// ---- OOPs/FB_HighLevelSystem.TcPOU
FUNCTION_BLOCK FB_HighLevelSystem IMPLEMENTS ITF_HighLevelSystem
VAR_INPUT
	eActivationStatus : ActivationStatus;
END_VAR
VAR_OUTPUT
END_VAR
VAR
END_VAR

PROPERTY eCondition : HighLevelCondition
GET
END_GET
END_PROPERTY

PROPERTY nErrorID : UDINT
GET
END_GET
END_PROPERTY

END_FUNCTION_BLOCK

// ---- POUs/ServiceModule/FB_DistanceSensor.TcPOU
FUNCTION_BLOCK FB_DistanceSensor IMPLEMENTS ITF_SubSystem
VAR_OUTPUT
	fDistance 			: LREAL;
END_VAR
VAR
	//Local
	fbEL6021			: FB_SerialComRS422;

	//ErrorBits
	bCommunicationError : BIT;
	bOutOfRange 		: BIT;
END_VAR
VAR CONSTANT
	fSMR 		: LREAL := 50.0;				// Start of Measuring Range
	fEMR 		: LREAL := 150.0;				// End of Measuring Range
END_VAR

fbEL6021(stReceiveData:=DistanceSensor.stEL6021In, stTransmitData:=DistanceSensor.stEL6021Out);

fDistance := fbEL6021.fDistance;

METHOD PRIVATE doCheckRange : BOOL
VAR_INPUT
	fDistanceValue : LREAL;
	fMax : LREAL;
	fMin : LREAL;
END_VAR
IF fDistanceValue < fMin OR fDistanceValue > fMax THEN
	doCheckRange := FALSE;
	fDistance := 999;
ELSE
	doCheckRange := TRUE;
END_IF
END_METHOD

PROPERTY eCondition : SubLevelCondition
GET
IF nErrorID <> 0 THEN
	eCondition := SubLevelCondition.ERROR;
ELSE
	eCondition := SubLevelCondition.RUN;
END_IF
END_GET
END_PROPERTY

PROPERTY nErrorID : UDINT
GET
IF fbEL6021.eReceiveErrorID <> COMERROR_NOERROR THEN
	bCommunicationError := TRUE;
ELSE
	bCommunicationError := FALSE;
END_IF

bOutOfRange := NOT doCheckRange(fDistanceValue:= fDistance, fMax:=fEMR, fMin:=fSMR);

nErrorID.0 := bCommunicationError;
nErrorID.1 := bOutOfRange;
END_GET
END_PROPERTY

END_FUNCTION_BLOCK

// ---- POUs/ServiceModule/DistanceSensor/FB_SerialComRS422.TcPOU
FUNCTION_BLOCK FB_SerialComRS422
VAR_IN_OUT
	stReceiveData 	: EL6inData22B;
	stTransmitData 	: EL6outData22B;
END_VAR
VAR_OUTPUT
	fDistance : LREAL;
	eReceiveErrorID	: ComError_t;
END_VAR
VAR
	//Receive Buffer
	fbEL6021Ctrl					: SerialLineControl;
	RxBuffer 						: ComBuffer;
	TxBuffer						: ComBuffer;
	//Receive Data
	fbReceiveByte					: ReceiveByte;				
	nFirstThreeBytesOfBuffer  		: ARRAY[0..2] OF BYTE;		// buffer storage for the three bytes that contain the distance information
	nRcvIndex						: UINT := 0;				// Counter
	nDistanceAsStringOfBits			: DINT;
END_VAR
VAR CONSTANT
	fSMR 		: LREAL := 50.0;				// Start of Measuring Range
	fEMR 		: LREAL := 150.0;				// End of Measuring Range
END_VAR

fbEL6021Ctrl(
			Mode:= SERIALLINEMODE_EL6_22B,
			pComIn:= ADR(stReceiveData),
			pComOut:= ADR(stTransmitData),
			SizeComIn:= SIZEOF(stReceiveData),
			Error=>,
			ErrorID=>,
			TxBuffer:=TxBuffer,
			RxBuffer:=RxBuffer,);

fbReceiveByte(RXbuffer := RxBuffer, Error => eReceiveErrorID);

WHILE fbReceiveByte.ByteReceived AND (nRcvIndex <= SIZEOF(nFirstThreeBytesOfBuffer)) DO
	fbReceiveByte(RXbuffer := RxBuffer);
	IF (fbReceiveByte.ReceivedByte.7) = 0 THEN
		nFirstThreeBytesOfBuffer[nRcvIndex] := fbReceiveByte.ReceivedByte;
		nRcvIndex := nRcvIndex + 1;
	ELSE
		nFirstThreeBytesOfBuffer[2] := fbReceiveByte.ReceivedByte;
		nRcvIndex	:= 0;
	END_IF
END_WHILE

doSortBits(nByteBuffer:=nFirstThreeBytesOfBuffer);
doConvertToDistanceValue(nBitString:=nDistanceAsStringOfBits, fMax:=fEMR, fMin:=fSMR);

METHOD PRIVATE doConvertToDistanceValue
VAR_INPUT
	nBitString : DINT;
	fMax : LREAL;
	fMIn : LREAL;
END_VAR
fDistance := 50.0 + 1.0/100.0 * (102.0/65520.0 * DINT_TO_LREAL(nBitString) - 1.0) * (fMax - fMIn);
END_METHOD

METHOD PRIVATE doSortBits
VAR_INPUT
	nByteBuffer : ARRAY [0..2] OF BYTE;
END_VAR
// Rearrange L,M,H Refer Pg 85. We seperate the distance bits from the error, transmissions, ect. -bits in this step.
// MemCopy is a possilbe way to simplify code. But since we need to work with bit and not buyts, this is actually the more readable code.
// Also TwinCAT demands CONST values when working with bit handeling, so loops are also not possible.
nDistanceAsStringOfBits.0 	:= nByteBuffer[0].0;
nDistanceAsStringOfBits.1 	:= nByteBuffer[0].1;
nDistanceAsStringOfBits.2 	:= nByteBuffer[0].2;
nDistanceAsStringOfBits.3 	:= nByteBuffer[0].3;
nDistanceAsStringOfBits.4 	:= nByteBuffer[0].4;
nDistanceAsStringOfBits.5 	:= nByteBuffer[0].5;
nDistanceAsStringOfBits.6 	:= nByteBuffer[1].0;
nDistanceAsStringOfBits.7 	:= nByteBuffer[1].1;
nDistanceAsStringOfBits.8 	:= nByteBuffer[1].2;
nDistanceAsStringOfBits.9 	:= nByteBuffer[1].3;
nDistanceAsStringOfBits.10 	:= nByteBuffer[1].4;
nDistanceAsStringOfBits.11	:= nByteBuffer[1].5;
nDistanceAsStringOfBits.12 	:= nByteBuffer[2].0;
nDistanceAsStringOfBits.13 	:= nByteBuffer[2].1;
nDistanceAsStringOfBits.14 	:= nByteBuffer[2].2;
nDistanceAsStringOfBits.15 	:= nByteBuffer[2].3;
END_METHOD

END_FUNCTION_BLOCK

// ---- POUs/ServiceModule/FB_BoxLED.TcPOU
FUNCTION_BLOCK FB_BoxLED IMPLEMENTS ITF_SubSystem
VAR_INPUT
	eMode : LEDMode;
END_VAR
VAR
	//Local
	nBoxLED : INT;
	fbFlashingTimer : TON;
	bOn : BOOL;
	
	aErrorTimer : ARRAY [0..1] OF TON;
	
	//ErrorBits
	bTemperatureTooHigh : BIT;
	bNoSupplyVoltage : BIT;
END_VAR
VAR CONSTANT
	nIntensity : INT := 32767;				//Intensity [0..32767]
	fDimFactor : REAL := 0.01;				//Percentage (0..100%)
	tSlowFlashingTime : TIME := T#1S;		
	tFastFlashingTime : TIME := T#100MS;
END_VAR

CASE eMode OF
	LEDMode.Off:
			doTurnOn(nBrightness := 0);
	LEDMode.On:
			doTurnOn(nBrightness := nIntensity);
	LEDMode.Dimmed:
			doDimming(fDimmingFactor:=fDimFactor);
	LEDMode.SlowFlashing:
			doFlashing(tFlashingTime:=tSlowFlashingTime);
	LEDMode.FastFlashing:
			doFlashing(tFlashingTime:=tFastFlashingTime);
END_CASE

doSetClampValues();
doGetClampValues();

METHOD PRIVATE doDimming
VAR_INPUT
	fDimmingFactor : REAL;
END_VAR
nBoxLED := REAL_TO_INT(fDimmingFactor * nIntensity);
END_METHOD

METHOD PRIVATE doFlashing
VAR_INPUT
	tFlashingTime : TIME;
END_VAR
fbFlashingTimer(IN:=TRUE, PT:=tFlashingTime);
IF fbFlashingTimer.Q THEN
	fbFlashingTimer(IN:=FALSE);
	bOn := NOT bOn;	
END_IF
IF bOn THEN
	nBoxLED := nIntensity;
ELSE
	nBoxLED := 0;
END_IF
END_METHOD

METHOD PRIVATE doGetClampValues
bTemperatureTooHigh := BoxLED.bBoxGreenWarning;
bNoSupplyVoltage := BoxLED.bBoxGreenError;
END_METHOD

METHOD PRIVATE doSetClampValues
BoxLED.nBoxGreen := nBoxLED;
END_METHOD

METHOD PRIVATE doTurnOn
VAR_INPUT
	nBrightness : INT;
END_VAR
nBoxLED := nBrightness;
END_METHOD

PROPERTY eCondition : SubLevelCondition
GET
IF nErrorID <> 0 THEN
	eCondition := SubLevelCondition.ERROR;
ELSE
	eCondition := SubLevelCondition.RUN;
END_IF
END_GET
END_PROPERTY

PROPERTY nErrorID : UDINT
GET
nErrorID.0 := aErrorTimer[0].Q;
nErrorID.1 := aErrorTimer[1].Q;

aErrorTimer[0](IN := bTemperatureTooHigh, PT := T#5S);
aErrorTimer[1](IN := bNoSupplyVoltage, PT := T#5S);
END_GET
END_PROPERTY

END_FUNCTION_BLOCK

// ---- POUs/ServiceModule/FB_RGBLED.TcPOU
FUNCTION_BLOCK FB_RGBLED IMPLEMENTS ITF_SubSystem
VAR_INPUT
	eColor : LEDColor;
END_VAR
VAR
	//Local
	nRedLED : INT;
	nGreenLED : INT;
	nBlueLED : INT;
	
	aErrorTimer : ARRAY [0..5] OF TON;
	
	//ErrorBits
	bRedTemperatureTooHigh : BIT;
	bRedNoSupplyVoltage : BIT;
	bGreenTemperatureTooHigh : BIT;
	bGreenNoSupplyVoltage : BIT;
	bBlueTemperatureTooHigh : BIT;
	bBlueNoSupplyVoltage : BIT;	
END_VAR
VAR CONSTANT
	nMax : INT := 32767;		//Maximum Intensity (100%)
	nMin : INT := 0;			//Off (0%)
END_VAR

CASE eColor OF
	LEDColor.Off:
		nRedLED := nMin;
		nGreenLED := nMin;
		nBlueLED := nMin;
	LEDColor.Red:
		nRedLED := nMax;
		nGreenLED := nMin;
		nBlueLED := nMin;
	LEDColor.Green:
		nRedLED := nMin;
		nGreenLED := nMax;
		nBlueLED := nMin;
	LEDColor.Blue:
		nRedLED := nMin;
		nGreenLED := nMin;
		nBlueLED := nMax;
END_CASE



doSetClampValues();
doGetClampValues();

METHOD PRIVATE doGetClampValues
VAR_INPUT
END_VAR
bRedTemperatureTooHigh := RGBLED.bRedWarning;
bRedNoSupplyVoltage := RGBLED.bRedError;
bGreenTemperatureTooHigh := RGBLED.bGreenWarning;
bGreenNoSupplyVoltage := RGBLED.bGreenError;
bBlueTemperatureTooHigh := RGBLED.bBlueWarning;
bBlueNoSupplyVoltage := RGBLED.bBlueError;
END_METHOD

METHOD PRIVATE doSetClampValues
RGBLED.nRed := nRedLED;
RGBLED.nGreen := nGreenLED;
RGBLED.nBlue := nBlueLED;
END_METHOD

PROPERTY eCondition : SubLevelCondition
GET
IF nErrorID <> 0 THEN
	eCondition := SubLevelCondition.ERROR;
ELSE
	eCondition := SubLevelCondition.RUN;
END_IF
END_GET
END_PROPERTY

PROPERTY nErrorID : UDINT
GET
nErrorID.0 := aErrorTimer[0].Q;
nErrorID.1 := aErrorTimer[1].Q;
nErrorID.2 := aErrorTimer[2].Q;
nErrorID.3 := aErrorTimer[3].Q;
nErrorID.4 := aErrorTimer[4].Q;
nErrorID.5 := aErrorTimer[5].Q;

aErrorTimer[0](IN:=bRedTemperatureTooHigh, PT:=T#5S);
aErrorTimer[1](IN:=bRedNoSupplyVoltage, PT:=T#5S);
aErrorTimer[2](IN:=bGreenTemperatureTooHigh, PT:=T#5S);
aErrorTimer[3](IN:=bGreenNoSupplyVoltage, PT:=T#5S);
aErrorTimer[4](IN:=bBlueTemperatureTooHigh, PT:=T#5S);
aErrorTimer[5](IN:=bBlueNoSupplyVoltage, PT:=T#5S);
END_GET
END_PROPERTY

END_FUNCTION_BLOCK

// ---- POUs/FB_LevitationSystem.TcPOU
FUNCTION_BLOCK FB_LevitationSystem EXTENDS FB_HighLevelSystem
VAR_INPUT
	eState : LevitationSystemSTM;
	nTGControlOption : USINT;
	//eActivationStatus : ActivationStatus;
END_VAR
VAR_OUTPUT
	bEnableCurrentController : BOOL;
	bEnableIControl : BOOL;
	bEnablePControl : BOOL;
END_VAR
VAR
	fbEqualizingControl			: FB_EqualizingController;
	fbTrajectoryGeneratorXMC1	: FB_TrajectoryGenerator;
	fbTrajectoryGeneratorXMC2	: FB_TrajectoryGenerator;
	fbTrajectoryGeneratorXMC3	: FB_TrajectoryGenerator;
	fbTrajectoryGeneratorXMC4	: FB_TrajectoryGenerator;
	
	fActualLevDistanceForFmag : ARRAY [0..3] OF REAL;
	fActualLevCurrentForFmag : ARRAY [0..3] OF REAL;
	
	fDesiredLevDistance : REAL;
END_VAR

IF eActivationStatus = ActivationStatus.Enabled THEN
	//High Level State Machine
	CASE eState OF
		LevitationSystemSTM.Idling:
			;
			
			
		LevitationSystemSTM.Stationary:
			bEnableCurrentController := FALSE;
			fbTrajectoryGeneratorXMC1.bTransition := FALSE;
			fbTrajectoryGeneratorXMC2.bTransition := FALSE;
			fbTrajectoryGeneratorXMC3.bTransition := FALSE;
			fbTrajectoryGeneratorXMC4.bTransition := FALSE;

			fbEqualizingControl.bActive := FALSE;		
		
			doSetOperationMode();
			
			fbTrajectoryGeneratorXMC1();
			fbTrajectoryGeneratorXMC2();
			fbTrajectoryGeneratorXMC3();
			fbTrajectoryGeneratorXMC4();
			fbEqualizingControl();
			
		LevitationSystemSTM.Transitioning:
			bEnableCurrentController := TRUE;
//			fbTrajectoryGeneratorXMC1.bTransition := TRUE;
//			fbTrajectoryGeneratorXMC2.bTransition := TRUE;
//			fbTrajectoryGeneratorXMC3.bTransition := TRUE;
//			fbTrajectoryGeneratorXMC4.bTransition := TRUE;
			
			//optional AirGap Check to go back into Transition		
			IF fActualLevDistanceForFmag[0] <> fDesiredLevDistance THEN
				fbTrajectoryGeneratorXMC1.bTransition := TRUE;
			ELSE
				fbTrajectoryGeneratorXMC1.bTransition := FALSE;
			END_IF
			IF fActualLevDistanceForFmag[1] <> fDesiredLevDistance THEN
				fbTrajectoryGeneratorXMC2.bTransition := TRUE;
			ELSE
				fbTrajectoryGeneratorXMC2.bTransition := FALSE;
			END_IF
			IF fActualLevDistanceForFmag[2] <> fDesiredLevDistance THEN
				fbTrajectoryGeneratorXMC3.bTransition := TRUE;
			ELSE
				fbTrajectoryGeneratorXMC3.bTransition := FALSE;
			END_IF
			IF fActualLevDistanceForFmag[3] <> fDesiredLevDistance THEN
				fbTrajectoryGeneratorXMC4.bTransition := TRUE;
			ELSE
				fbTrajectoryGeneratorXMC4.bTransition := FALSE;
			END_IF
			
			fbEqualizingControl.bActive := FALSE;
			
			fbTrajectoryGeneratorXMC1();
			fbTrajectoryGeneratorXMC2();
			fbTrajectoryGeneratorXMC3();
			fbTrajectoryGeneratorXMC4();
			fbEqualizingControl();
			
			
		LevitationSystemSTM.HoldingAirGap:
			bEnableCurrentController := FALSE;
			fbTrajectoryGeneratorXMC1.bTransition := FALSE;
			fbTrajectoryGeneratorXMC2.bTransition := FALSE;
			fbTrajectoryGeneratorXMC3.bTransition := FALSE;
			fbTrajectoryGeneratorXMC4.bTransition := FALSE;
			
			fbEqualizingControl.bActive := TRUE;
			
			doCalculateFmagValuesForEC(	fActualLevDistance := fActualLevDistanceForFmag,			//to be implemented
										fActualCurrent := fActualLevCurrentForFmag);
			
			fbTrajectoryGeneratorXMC1();
			fbTrajectoryGeneratorXMC2();
			fbTrajectoryGeneratorXMC3();
			fbTrajectoryGeneratorXMC4();
			fbEqualizingControl();
			
			
		LevitationSystemSTM.TransitioningToZero:
			bEnableCurrentController := TRUE;
			fbTrajectoryGeneratorXMC1.bTransition := TRUE;
			fbTrajectoryGeneratorXMC2.bTransition := TRUE;
			fbTrajectoryGeneratorXMC3.bTransition := TRUE;
			fbTrajectoryGeneratorXMC4.bTransition := TRUE;
			
			fbEqualizingControl.bActive := FALSE;
			
			doSetPresetTGValuesForBackToGround();		//to be implemented with Controller structure
			
			fbTrajectoryGeneratorXMC1();
			fbTrajectoryGeneratorXMC2();
			fbTrajectoryGeneratorXMC3();
			fbTrajectoryGeneratorXMC4();
			fbEqualizingControl();
			
	END_CASE	

END_IF

PROPERTY PUBLIC aECOutputZVector : ARRAY [0..3] OF REAL
GET
aECOutputZVector[0] := fbEqualizingControl.fdzVector[0];
aECOutputZVector[1] := fbEqualizingControl.fdzVector[1];
aECOutputZVector[2] := fbEqualizingControl.fdzVector[2];
aECOutputZVector[3] := fbEqualizingControl.fdzVector[3];
END_GET
END_PROPERTY

PROPERTY PUBLIC aTGActualLevAcceleration : ARRAY [0..3] OF REAL
SET
fbTrajectoryGeneratorXMC1.fInitialAcceleration := aTGActualLevAcceleration[0];
fbTrajectoryGeneratorXMC2.fInitialAcceleration := aTGActualLevAcceleration[1];
fbTrajectoryGeneratorXMC3.fInitialAcceleration := aTGActualLevAcceleration[2];
fbTrajectoryGeneratorXMC4.fInitialAcceleration := aTGActualLevAcceleration[3];
END_SET
END_PROPERTY

PROPERTY PUBLIC aTGActualLevCurrent : ARRAY [0..3] OF REAL
SET
fActualLevCurrentForFmag := aTGActualLevCurrent;

fbTrajectoryGeneratorXMC1.fInitialCurrent := aTGActualLevCurrent[0];
fbTrajectoryGeneratorXMC2.fInitialCurrent := aTGActualLevCurrent[1];
fbTrajectoryGeneratorXMC3.fInitialCurrent := aTGActualLevCurrent[2];
fbTrajectoryGeneratorXMC4.fInitialCurrent := aTGActualLevCurrent[3];
END_SET
END_PROPERTY

PROPERTY PUBLIC aTGActualLevDistance : ARRAY [0..3] OF REAL
SET
fActualLevDistanceForFmag := aTGActualLevDistance;

fbTrajectoryGeneratorXMC1.fInitialAirGap := aTGActualLevDistance[0];
fbTrajectoryGeneratorXMC2.fInitialAirGap := aTGActualLevDistance[1];
fbTrajectoryGeneratorXMC3.fInitialAirGap := aTGActualLevDistance[2];
fbTrajectoryGeneratorXMC4.fInitialAirGap := aTGActualLevDistance[3];
END_SET
END_PROPERTY

PROPERTY PUBLIC aTGActualLevVelocity : ARRAY [0..3] OF REAL
SET
fbTrajectoryGeneratorXMC1.fInitialVelocity := aTGActualLevVelocity[0];
fbTrajectoryGeneratorXMC2.fInitialVelocity := aTGActualLevVelocity[1];
fbTrajectoryGeneratorXMC3.fInitialVelocity := aTGActualLevVelocity[2];
fbTrajectoryGeneratorXMC4.fInitialVelocity := aTGActualLevVelocity[3];
END_SET
END_PROPERTY

PROPERTY PUBLIC aTGOutputLevAcceleration : ARRAY [0..3] OF REAL
GET
aTGOutputLevAcceleration[0] := fbTrajectoryGeneratorXMC1.fNewReferenceValueForAcceleration;
aTGOutputLevAcceleration[1] := fbTrajectoryGeneratorXMC2.fNewReferenceValueForAcceleration;
aTGOutputLevAcceleration[2] := fbTrajectoryGeneratorXMC3.fNewReferenceValueForAcceleration;
aTGOutputLevAcceleration[3] := fbTrajectoryGeneratorXMC4.fNewReferenceValueForAcceleration;
END_GET
END_PROPERTY

PROPERTY PUBLIC aTGOutputLevCurrent : ARRAY [0..3] OF REAL
GET
aTGOutputLevCurrent[0] := fbTrajectoryGeneratorXMC1.fNewReferenceValueForCurrent;
aTGOutputLevCurrent[1] := fbTrajectoryGeneratorXMC2.fNewReferenceValueForCurrent;
aTGOutputLevCurrent[2] := fbTrajectoryGeneratorXMC3.fNewReferenceValueForCurrent;
aTGOutputLevCurrent[3] := fbTrajectoryGeneratorXMC4.fNewReferenceValueForCurrent;
END_GET
END_PROPERTY

PROPERTY PUBLIC aTGOutputLevDistance : ARRAY [0..3] OF REAL
GET
aTGOutputLevDistance[0] := fbTrajectoryGeneratorXMC1.fNewReferenceValueForAirGap;
aTGOutputLevDistance[1] := fbTrajectoryGeneratorXMC2.fNewReferenceValueForAirGap;
aTGOutputLevDistance[2] := fbTrajectoryGeneratorXMC3.fNewReferenceValueForAirGap;
aTGOutputLevDistance[3] := fbTrajectoryGeneratorXMC4.fNewReferenceValueForAirGap;
END_GET
END_PROPERTY

PROPERTY PUBLIC aTGOutputLevForce : ARRAY [0..3] OF REAL
GET
aTGOutputLevForce[0] := fbTrajectoryGeneratorXMC1.fNewReferenceValueForForce;
aTGOutputLevForce[1] := fbTrajectoryGeneratorXMC2.fNewReferenceValueForForce;
aTGOutputLevForce[2] := fbTrajectoryGeneratorXMC3.fNewReferenceValueForForce;
aTGOutputLevForce[3] := fbTrajectoryGeneratorXMC4.fNewReferenceValueForForce;
END_GET
END_PROPERTY

PROPERTY PUBLIC aTGOutputLevVelocity : ARRAY [0..3] OF REAL
GET
aTGOutputLevVelocity[0] := fbTrajectoryGeneratorXMC1.fNewReferenceVaueForVelocity;
aTGOutputLevVelocity[1] := fbTrajectoryGeneratorXMC2.fNewReferenceVaueForVelocity;
aTGOutputLevVelocity[2] := fbTrajectoryGeneratorXMC3.fNewReferenceVaueForVelocity;
aTGOutputLevVelocity[3] := fbTrajectoryGeneratorXMC4.fNewReferenceVaueForVelocity;
END_GET
END_PROPERTY

PROPERTY PUBLIC aTGOutputLevVoltage : ARRAY [0..3] OF REAL
GET
aTGOutputLevVoltage[0] := fbTrajectoryGeneratorXMC1.fNewReferenceValueForVoltage;
aTGOutputLevVoltage[1] := fbTrajectoryGeneratorXMC2.fNewReferenceValueForVoltage;
aTGOutputLevVoltage[2] := fbTrajectoryGeneratorXMC3.fNewReferenceValueForVoltage;
aTGOutputLevVoltage[3] := fbTrajectoryGeneratorXMC4.fNewReferenceValueForVoltage;
END_GET
END_PROPERTY

PROPERTY PUBLIC bTrajectoryCompleted : BOOL
GET
VAR
	bTrajectoryCompletedXMC1 : BOOL;
	bTrajectoryCompletedXMC2 : BOOL;
	bTrajectoryCompletedXMC3 : BOOL;
	bTrajectoryCompletedXMC4 : BOOL;
END_VAR
bTrajectoryCompletedXMC1 := fbTrajectoryGeneratorXMC1.bTrajectoryCompleted;
bTrajectoryCompletedXMC2 := fbTrajectoryGeneratorXMC2.bTrajectoryCompleted;
bTrajectoryCompletedXMC3 := fbTrajectoryGeneratorXMC3.bTrajectoryCompleted;
bTrajectoryCompletedXMC4 := fbTrajectoryGeneratorXMC4.bTrajectoryCompleted;

IF bTrajectoryCompletedXMC1 AND bTrajectoryCompletedXMC2 AND bTrajectoryCompletedXMC3 AND bTrajectoryCompletedXMC4 THEN
	bTrajectoryCompleted := TRUE;
ELSE
	bTrajectoryCompleted := FALSE;
END_IF
END_GET
END_PROPERTY

METHOD PRIVATE doCalculateFmagValuesForEC
VAR_INPUT
	fActualLevDistance : ARRAY [0..3] OF REAL;
	fActualCurrent		: ARRAY [0..3] OF REAL;
END_VAR
fbEqualizingControl.fActualDeltaFmag := 0;
END_METHOD

METHOD PRIVATE doSetOperationMode
VAR_INPUT
END_VAR
IF nTGControlOption.0 THEN
	fbTrajectoryGeneratorXMC1.eMode := TGControllerMode.IControl;
	fbTrajectoryGeneratorXMC2.eMode := TGControllerMode.IControl;
	fbTrajectoryGeneratorXMC3.eMode := TGControllerMode.IControl;
	fbTrajectoryGeneratorXMC4.eMode := TGControllerMode.IControl;
	
	bEnableIControl := TRUE;
	bEnablePControl := FALSE;
END_IF

IF nTGControlOption.1 THEN
	fbTrajectoryGeneratorXMC1.eMode := TGControllerMode.PControl;
	fbTrajectoryGeneratorXMC2.eMode := TGControllerMode.PControl;
	fbTrajectoryGeneratorXMC3.eMode := TGControllerMode.PControl;
	fbTrajectoryGeneratorXMC4.eMode := TGControllerMode.PControl;
	
	bEnableIControl := FALSE;
	bEnablePControl := TRUE;
END_IF
END_METHOD

METHOD PRIVATE doSetPresetTGValuesForBackToGround
VAR_INPUT
END_VAR
END_METHOD

PROPERTY eCondition : HighLevelCondition
GET
IF eActivationStatus = ActivationStatus.Disabled THEN
	eCondition := HighLevelCondition.SLEEP;
ELSE
	IF fbTrajectoryGeneratorXMC1.eCondition = SubLevelCondition.RUN AND fbTrajectoryGeneratorXMC2.eCondition = SubLevelCondition.RUN AND fbTrajectoryGeneratorXMC3.eCondition = SubLevelCondition.RUN AND fbTrajectoryGeneratorXMC4.eCondition = SubLevelCondition.RUN AND fbEqualizingControl.eCondition = SubLevelCondition.RUN THEN
		eCondition := HighLevelCondition.RUN;
	ELSE
		eCondition := HighLevelCondition.INIT;
	END_IF
END_IF
END_GET
END_PROPERTY

PROPERTY PUBLIC fTGDesiredLevAcceleration : REAL
SET
fbTrajectoryGeneratorXMC1.fDesiredAccelerationAfterTransitioning := fTGDesiredLevAcceleration;
fbTrajectoryGeneratorXMC2.fDesiredAccelerationAfterTransitioning := fTGDesiredLevAcceleration;
fbTrajectoryGeneratorXMC3.fDesiredAccelerationAfterTransitioning := fTGDesiredLevAcceleration;
fbTrajectoryGeneratorXMC4.fDesiredAccelerationAfterTransitioning := fTGDesiredLevAcceleration;
END_SET
END_PROPERTY

PROPERTY PUBLIC fTGDesiredLevDistance : REAL
SET
fbTrajectoryGeneratorXMC1.fDesiredAirGapAfterTransitioning := fTGDesiredLevDistance;
fbTrajectoryGeneratorXMC2.fDesiredAirGapAfterTransitioning := fTGDesiredLevDistance;
fbTrajectoryGeneratorXMC3.fDesiredAirGapAfterTransitioning := fTGDesiredLevDistance;
fbTrajectoryGeneratorXMC4.fDesiredAirGapAfterTransitioning := fTGDesiredLevDistance;

fDesiredLevDistance := fTGDesiredLevDistance;
END_SET
END_PROPERTY

PROPERTY PUBLIC fTGDesiredLevTime : REAL
SET
fbTrajectoryGeneratorXMC1.tDesiredTimeForTransitioning := REAL_TO_TIME(fTGDesiredLevTime);
fbTrajectoryGeneratorXMC2.tDesiredTimeForTransitioning := REAL_TO_TIME(fTGDesiredLevTime);
fbTrajectoryGeneratorXMC3.tDesiredTimeForTransitioning := REAL_TO_TIME(fTGDesiredLevTime);
fbTrajectoryGeneratorXMC4.tDesiredTimeForTransitioning := REAL_TO_TIME(fTGDesiredLevTime);
END_SET
END_PROPERTY

PROPERTY PUBLIC fTGDesiredLevVelocity : REAL
SET
fbTrajectoryGeneratorXMC1.fDesiredVelocityAfterTransitioning := fTGDesiredLevVelocity;
fbTrajectoryGeneratorXMC2.fDesiredVelocityAfterTransitioning := fTGDesiredLevVelocity;
fbTrajectoryGeneratorXMC3.fDesiredVelocityAfterTransitioning := fTGDesiredLevVelocity;
fbTrajectoryGeneratorXMC4.fDesiredVelocityAfterTransitioning := fTGDesiredLevVelocity;
END_SET
END_PROPERTY

PROPERTY nErrorID : UDINT
GET
VAR
	nErrorBitsTG1 : UDINT;
	nErrorBitsTG2 : UDINT;
	nErrorBitsTG3 : UDINT;
	nErrorBitsTG4 : UDINT;
	nErrorBitsEC	: UDINT;
END_VAR
nErrorBitsTG1 := fbTrajectoryGeneratorXMC1.nErrorID;
nErrorBitsTG2 := fbTrajectoryGeneratorXMC2.nErrorID;
nErrorBitsTG3 := fbTrajectoryGeneratorXMC3.nErrorID;
nErrorBitsTG4 := fbTrajectoryGeneratorXMC4.nErrorID;
nErrorBitsEC := fbEqualizingControl.nErrorID;


nErrorID.0 := nErrorBitsEC.0;
nErrorID.1 := nErrorBitsEC.1;
nErrorID.2 := nErrorBitsTG1.0;
nErrorID.3 := nErrorBitsTG1.1;
nErrorID.4 := nErrorBitsTG1.2;
nErrorID.5 := nErrorBitsTG1.3;
nErrorID.6 := nErrorBitsTG1.4;
nErrorID.7 := nErrorBitsTG1.5;
nErrorID.8 := nErrorBitsTG2.0;
nErrorID.9 := nErrorBitsTG2.1;
nErrorID.10 := nErrorBitsTG2.2;
nErrorID.11 := nErrorBitsTG2.3;
nErrorID.12 := nErrorBitsTG2.4;
nErrorID.13 := nErrorBitsTG2.5;
nErrorID.14 := nErrorBitsTG3.0;
nErrorID.15 := nErrorBitsTG3.1;
nErrorID.16 := nErrorBitsTG3.2;
nErrorID.17 := nErrorBitsTG3.3;
nErrorID.18 := nErrorBitsTG3.4;
nErrorID.19 := nErrorBitsTG3.5;
nErrorID.20 := nErrorBitsTG4.0;
nErrorID.21 := nErrorBitsTG4.1;
nErrorID.22 := nErrorBitsTG4.2;
nErrorID.23 := nErrorBitsTG4.3;
nErrorID.24 := nErrorBitsTG4.4;
nErrorID.25 := nErrorBitsTG4.5;
END_GET
END_PROPERTY

END_FUNCTION_BLOCK

// ---- POUs/Levitation/FB_EqualizingController.TcPOU
FUNCTION_BLOCK FB_EqualizingController IMPLEMENTS ITF_SubSystem
VAR_INPUT
	fActualDeltaFmag : REAL;
	bActive : BOOL;
END_VAR
VAR_OUTPUT 
	fdzVector : ARRAY [0..3] OF REAL;
END_VAR
VAR
	//Local
	fbPIDController : FB_BasicPID;
	fPIDOutput : LREAL;
	nPIDErrorID : UINT;

	//Error Bits
	bInvalidParamters : BIT;
	bInvalidCycleTime : BIT;
END_VAR
VAR CONSTANT
	//PID paramters
	fSetpointValue : REAL := 0; 			// Reference delta F = 0 N
	fCtrlCycleTime : REAL := 0.1; 			// Update cycle time of PID block
	fKp : REAL := 0.001;  					// Proportional gain of PID block
	fTn : REAL := 1/INT_TO_REAL(150); 
	fTv : REAL := 0;
	fTd : REAL := 0;
	//Saturation parameters
	fdzMax : REAL := 0.001;
	fdzMin : REAL := -0.001;
END_VAR

IF bActive THEN
	fbPIDController(fSetpointValue := fSetpointValue,
					fActualValue := fActualDeltaFmag,
					bReset := NOT bActive,
					fCtrlCycleTime := fCtrlCycleTime,
					fKp := fKp,
					fTn := fTn,
					fTv := fTv,
					fTd := fTd,
					fCtrlOutput => fPIDOutput, nErrorStatus => nPIDErrorID);

					
	// Update the dz output vector
	fdzVector[0] := (-1/INT_TO_REAL(7900))* LREAL_TO_REAL(fPIDOutput);
	fdzVector[1] := (1/INT_TO_REAL(7900))* LREAL_TO_REAL(fPIDOutput);
	fdzVector[2] := (-1/INT_TO_REAL(7900))* LREAL_TO_REAL(fPIDOutput);
	fdzVector[3] := (1/INT_TO_REAL(7900))* LREAL_TO_REAL(fPIDOutput);	  
	
	
	// Saturate the dz output vector
	IF fdzVector[0] > fdzMax THEN
		fdzVector[0] := fdzMax;
	ELSIF fdzVector[0] < fdzMin THEN
		fdzVector[0] := fdzMin;
	END_IF
	
	IF fdzVector[1] > fdzMax THEN
		fdzVector[1] := fdzMax;
	ELSIF fdzVector[1] < fdzMin THEN
		fdzVector[1] := fdzMin;
	END_IF
	
	IF fdzVector[2] > fdzMax THEN
		fdzVector[2] := fdzMax;
	ELSIF fdzVector[2] < fdzMin THEN
		fdzVector[2] := fdzMin;
	END_IF
	
	IF fdzVector[3] > fdzMax THEN
		fdzVector[3] := fdzMax;
	ELSIF fdzVector[3] < fdzMin THEN
		fdzVector[3] := fdzMin;
	END_IF
	
ELSE
	fdzVector[0] := 0;
	fdzVector[1] := 0;
	fdzVector[2] := 0;
	fdzVector[3] := 0;
END_IF

PROPERTY eCondition : SubLevelCondition
GET
IF nErrorID <> 0 THEN
	eCondition := SubLevelCondition.ERROR;
ELSE
	eCondition := SubLevelCondition.RUN;
END_IF
END_GET
END_PROPERTY

PROPERTY nErrorID : UDINT
GET
CASE nPIDErrorID OF
	0: 	bInvalidCycleTime := FALSE;
		bInvalidParamters := FALSE;
	1:	bInvalidParamters := TRUE;
	2:	bInvalidCycleTime := TRUE;
END_CASE
nErrorID.0 := bInvalidParamters;
nErrorID.1 := bInvalidCycleTime;
END_GET
END_PROPERTY

END_FUNCTION_BLOCK

// ---- POUs/Levitation/FB_TrajectoryGenerator.TcPOU
FUNCTION_BLOCK FB_TrajectoryGenerator IMPLEMENTS ITF_SubSystem
VAR_INPUT
	eMode : TGControllerMode;
	
	bTransition : BOOL;

	fInitialAirGap : REAL;
	fInitialVelocity : REAL;
	fInitialAcceleration : REAL;
	fInitialCurrent	: REAL;
	
	fDesiredAirGapAfterTransitioning : REAL;
	fDesiredVelocityAfterTransitioning : REAL;
	fDesiredAccelerationAfterTransitioning : REAL;
	tDesiredTimeForTransitioning : TIME;
END_VAR
VAR_OUTPUT
	fNewReferenceValueForAirGap : REAL;
	fNewReferenceVaueForVelocity : REAL;
	fNewReferenceValueForAcceleration : REAL;
	fNewReferenceValueForCurrent : REAL;
	fNewReferenceValueForVoltage : REAL;
	fNewReferenceValueForForce : REAL;
	
	bTrajectoryCompleted : BOOL;
END_VAR
VAR
	nCounter : UDINT;
	fbTransitionTimer : TON;
	tElapsedTransitionTime : TIME;

	//ErrorBits
	bAirGapValueOutOfRange : BOOL;
	bVelocityOutOfRange : BOOL;
	bAccelerationOutOfRange : BOOL;
	bCurrentOutOfRange : BOOL;
	bVoltageOutOfRange : BOOL;
	bForceOutOfRange : BOOL;
END_VAR
VAR CONSTANT
	nCounterMax : UDINT := 255;
	nCounterReset : UDINT := 2;
END_VAR

IF bTransition THEN
	nCounter := nCounter + 1;
	IF nCounter > nCounterMax THEN
		nCounter := nCounterReset;
	END_IF	

	CASE eMode OF
		TGControllerMode.IControl:
		IF nCounter = 1 THEN
			doSetInitialValues(	fInitialDistance := fInitialAirGap,				//BlackBox to be implemented with Controller structure
								fInitialVelocity := fInitialVelocity,
								fInitialAcceleration := fInitialAcceleration,
								fInitialCurrent := fInitialCurrent);
									
			doSetDesiredValues(	fDesiredDistance := fDesiredAirGapAfterTransitioning, 		//BlackBox to be implemented with Controller structure
								fDesiredVelocity := fDesiredVelocityAfterTransitioning,
								fDesiredAcceleration := fDesiredAccelerationAfterTransitioning,
								tDesiredTime := tDesiredTimeForTransitioning);		
			doCalculateTrajectory();										//BlackBox to be implemented with Controller structure
			
			fbTransitionTimer(IN := TRUE, PT := tDesiredTimeForTransitioning, ET => tElapsedTransitionTime);
		END_IF
		doGetTrajectoryValues(tElapsedTime := tElapsedTransitionTime);		//BlackBox to be implemented with Controller structure
		IF fbTransitionTimer.Q THEN
			bTrajectoryCompleted := TRUE;
		ELSE
			bTrajectoryCompleted := FALSE;
		END_IF
	
	
		TGControllerMode.PControl:
		IF nCounter = 1 THEN
			doSetInitialValues(	fInitialDistance := fInitialAirGap,				//BlackBox to be implemented with Controller structure
								fInitialVelocity := fInitialVelocity,
								fInitialAcceleration := fInitialAcceleration,
								fInitialCurrent := fInitialCurrent);
									
			doSetDesiredValues(	fDesiredDistance := fDesiredAirGapAfterTransitioning, 		//BlackBox to be implemented with Controller structure
								fDesiredVelocity := fDesiredVelocityAfterTransitioning,
								fDesiredAcceleration := fDesiredAccelerationAfterTransitioning,
								tDesiredTime := tDesiredTimeForTransitioning);		
			doCalculateTrajectory();										//BlackBox to be implemented with Controller structure
			
			fbTransitionTimer(IN := TRUE, PT := tDesiredTimeForTransitioning, ET => tElapsedTransitionTime);
		END_IF
		doGetTrajectoryValues(tElapsedTime := tElapsedTransitionTime);		//BlackBox to be implemented with Controller structure
		IF fbTransitionTimer.Q THEN
			bTrajectoryCompleted := TRUE;
		ELSE
			bTrajectoryCompleted := FALSE;
		END_IF
	END_CASE
ELSE
	nCounter := 0;
	fbTransitionTimer(IN := FALSE);
	
	bTrajectoryCompleted := TRUE;
	
	fNewReferenceValueForAirGap := 0;
	fNewReferenceVaueForVelocity := 0;
	fNewReferenceValueForAcceleration := 0;
	fNewReferenceValueForCurrent := 0;
	fNewReferenceValueForVoltage := 0;
	fNewReferenceValueForForce := 0;
END_IF

METHOD PRIVATE doCalculateTrajectory
VAR_INPUT
END_VAR
END_METHOD

METHOD PRIVATE doGetTrajectoryValues
VAR_INPUT
	tElapsedTime : TIME;
END_VAR
fNewReferenceValueForAirGap := 0;
fNewReferenceVaueForVelocity := 0;
fNewReferenceValueForAcceleration := 0;
fNewReferenceValueForCurrent := 0;
fNewReferenceValueForVoltage := 0;
fNewReferenceValueForForce := 0;
END_METHOD

METHOD PRIVATE doSetDesiredValues
VAR_INPUT
	fDesiredDistance : REAL;
	fDesiredVelocity : REAL;
	fDesiredAcceleration : REAL;
	tDesiredTime : TIME;
END_VAR
END_METHOD

METHOD PRIVATE doSetInitialValues
VAR_INPUT
	fInitialDistance : REAL;
	fInitialVelocity : REAL;
	fInitialAcceleration : REAL;
	fInitialCurrent : REAL;
END_VAR
END_METHOD

PROPERTY eCondition : SubLevelCondition
GET
IF nErrorID <> 0 THEN
	eCondition := SubLevelCondition.ERROR;
ELSE
	eCondition := SubLevelCondition.RUN;
END_IF
END_GET
END_PROPERTY

PROPERTY nErrorID : UDINT
GET
//*RangeAbfrage to be implemented*
bAirGapValueOutOfRange := FALSE;
bVelocityOutOfRange := FALSE;
bAccelerationOutOfRange := FALSE;
bCurrentOutOfRange := FALSE;
bVoltageOutOfRange := FALSE;
bForceOutOfRange := FALSE;

nErrorID.0 := bAirGapValueOutOfRange;
nErrorID.1 := bVelocityOutOfRange;
nErrorID.2 := bAccelerationOutOfRange;
nErrorID.3 := bCurrentOutOfRange;
nErrorID.4 := bVoltageOutOfRange;
nErrorID.5 := bForceOutOfRange;
END_GET
END_PROPERTY

END_FUNCTION_BLOCK

// ---- POUs/FB_GuidanceSystem.TcPOU
FUNCTION_BLOCK FB_GuidanceSystem EXTENDS FB_HighLevelSystem
VAR_INPUT
	eState : GuidanceSystemSTM;
	nGCControlOption : USINT;
	//eActivationStatus : ActivationStatus;
END_VAR
VAR
	fbAccelerationSensor1 : FB_AccelerationSensor;
	fbAccelerationSensor2 : FB_AccelerationSensor;
	fbGuidanceControllerXMC1 : FB_GuidanceController;
	fbGuidanceControllerXMC2 : FB_GuidanceController;
	fbGuidanceControllerXMC3 : FB_GuidanceController;
	fbGuidanceControllerXMC4 : FB_GuidanceController;
END_VAR
VAR_OUTPUT
	bEnableCurrentController : BOOL;
	bEnableIControl			: BOOL;
	bEnablePControl			: BOOL;
END_VAR

IF eActivationStatus = ActivationStatus.Enabled THEN
	//High Level State Machine
	CASE eState OF
		GuidanceSystemSTM.Idling:
				fbAccelerationSensor1(stRS232Inputs:=AccelerationSensor.stEL6001InIMU1, stRS232Outputs:=AccelerationSensor.stEL6001OutIMU1);
				fbAccelerationSensor2(stRS232Inputs:=AccelerationSensor.stEL6001InIMU2, stRS232Outputs:=AccelerationSensor.stEL6001OutIMU2);
		
		GuidanceSystemSTM.PreRunning:
				bEnableCurrentController := FALSE;
				fbGuidanceControllerXMC1.bActive := FALSE;
				fbGuidanceControllerXMC2.bActive := FALSE;
				fbGuidanceControllerXMC3.bActive := FALSE;
				fbGuidanceControllerXMC4.bActive := FALSE;
				
				doSetOperationMode();

				fbAccelerationSensor1(stRS232Inputs:=AccelerationSensor.stEL6001InIMU1, stRS232Outputs:=AccelerationSensor.stEL6001OutIMU1);
				fbAccelerationSensor2(stRS232Inputs:=AccelerationSensor.stEL6001InIMU2, stRS232Outputs:=AccelerationSensor.stEL6001OutIMU2);
				fbGuidanceControllerXMC1();
				fbGuidanceControllerXMC2();
				fbGuidanceControllerXMC3();
				fbGuidanceControllerXMC4();	
		
		
		GuidanceSystemSTM.Running:
				bEnableCurrentController := TRUE;
				fbGuidanceControllerXMC1.bActive := TRUE;
				fbGuidanceControllerXMC2.bActive := TRUE;
				fbGuidanceControllerXMC3.bActive := TRUE;
				fbGuidanceControllerXMC4.bActive := TRUE;

				fbAccelerationSensor1(stRS232Inputs:=AccelerationSensor.stEL6001InIMU1, stRS232Outputs:=AccelerationSensor.stEL6001OutIMU1);
				fbAccelerationSensor2(stRS232Inputs:=AccelerationSensor.stEL6001InIMU2, stRS232Outputs:=AccelerationSensor.stEL6001OutIMU2);
				fbGuidanceControllerXMC1();
				fbGuidanceControllerXMC2();
				fbGuidanceControllerXMC3();
				fbGuidanceControllerXMC4();		

		GuidanceSystemSTM.PostRunning:
				bEnableCurrentController := FALSE;
				fbGuidanceControllerXMC1.bActive := FALSE;
				fbGuidanceControllerXMC2.bActive := FALSE;
				fbGuidanceControllerXMC3.bActive := FALSE;
				fbGuidanceControllerXMC4.bActive := FALSE;
				
				fbAccelerationSensor1(stRS232Inputs:=AccelerationSensor.stEL6001InIMU1, stRS232Outputs:=AccelerationSensor.stEL6001OutIMU1);
				fbAccelerationSensor2(stRS232Inputs:=AccelerationSensor.stEL6001InIMU2, stRS232Outputs:=AccelerationSensor.stEL6001OutIMU2);
				fbGuidanceControllerXMC1();
				fbGuidanceControllerXMC2();
				fbGuidanceControllerXMC3();
				fbGuidanceControllerXMC4();			
	END_CASE
END_IF

PROPERTY PUBLIC aGCActualGuidAcceleration : ARRAY [0..3] OF REAL
SET
fbGuidanceControllerXMC1.fActualYAcceleration := aGCActualGuidAcceleration[0];
fbGuidanceControllerXMC2.fActualYAcceleration := aGCActualGuidAcceleration[1];
fbGuidanceControllerXMC3.fActualYAcceleration := aGCActualGuidAcceleration[2];
fbGuidanceControllerXMC4.fActualYAcceleration := aGCActualGuidAcceleration[3];
END_SET
END_PROPERTY

PROPERTY PUBLIC aGCActualGuidCurrent : ARRAY [0..3] OF REAL
SET
fbGuidanceControllerXMC1.fActualCurrent := aGCActualGuidCurrent[0];
fbGuidanceControllerXMC2.fActualCurrent := aGCActualGuidCurrent[1];
fbGuidanceControllerXMC3.fActualCurrent := aGCActualGuidCurrent[2];
fbGuidanceControllerXMC4.fActualCurrent := aGCActualGuidCurrent[3];
END_SET
END_PROPERTY

PROPERTY PUBLIC aGCActualGuidDistance : ARRAY [0..3] OF REAL
SET
fbGuidanceControllerXMC1.fActualYDistance := aGCActualGuidDistance[0];
fbGuidanceControllerXMC2.fActualYDistance := aGCActualGuidDistance[1];
fbGuidanceControllerXMC3.fActualYDistance := aGCActualGuidDistance[2];
fbGuidanceControllerXMC4.fActualYDistance := aGCActualGuidDistance[3];
END_SET
END_PROPERTY

PROPERTY PUBLIC aGCOutputGuidCurrent : ARRAY [0..3] OF REAL
GET
aGCOutputGuidCurrent[0] := fbGuidanceControllerXMC1.fNewReferenceValueForCurrent;
aGCOutputGuidCurrent[1] := fbGuidanceControllerXMC2.fNewReferenceValueForCurrent;
aGCOutputGuidCurrent[2] := fbGuidanceControllerXMC3.fNewReferenceValueForCurrent;
aGCOutputGuidCurrent[3] := fbGuidanceControllerXMC4.fNewReferenceValueForCurrent;
END_GET
END_PROPERTY

PROPERTY PUBLIC aGCOutputGuidForce : ARRAY [0..3] OF REAL
GET
aGCOutputGuidForce[0] := fbGuidanceControllerXMC1.fNewRefrenceValueForForce;
aGCOutputGuidForce[1] := fbGuidanceControllerXMC2.fNewRefrenceValueForForce;
aGCOutputGuidForce[2] := fbGuidanceControllerXMC3.fNewRefrenceValueForForce;
aGCOutputGuidForce[3] := fbGuidanceControllerXMC4.fNewRefrenceValueForForce;
END_GET
END_PROPERTY

PROPERTY PUBLIC aGCOutputGuidVoltage : ARRAY [0..3] OF REAL
GET
aGCOutputGuidVoltage[0] := fbGuidanceControllerXMC1.fNewreferenceValueForVoltage;
aGCOutputGuidVoltage[1] := fbGuidanceControllerXMC2.fNewreferenceValueForVoltage;
aGCOutputGuidVoltage[2] := fbGuidanceControllerXMC3.fNewreferenceValueForVoltage;
aGCOutputGuidVoltage[3] := fbGuidanceControllerXMC4.fNewreferenceValueForVoltage;
END_GET
END_PROPERTY

PROPERTY PUBLIC aGCReferenceYSignal : REAL
SET
fbGuidanceControllerXMC1.fDesiredDeviationFromCenterLine := aGCReferenceYSignal;
fbGuidanceControllerXMC2.fDesiredDeviationFromCenterLine := aGCReferenceYSignal;
fbGuidanceControllerXMC3.fDesiredDeviationFromCenterLine := aGCReferenceYSignal;
fbGuidanceControllerXMC4.fDesiredDeviationFromCenterLine := aGCReferenceYSignal;
END_SET
END_PROPERTY

PROPERTY aIMU1Acceleration : ARRAY [0..2] OF REAL
GET
aIMU1Acceleration := fbAccelerationSensor1.aAccelerationValues;
END_GET
END_PROPERTY

PROPERTY aIMU2Acceleration : ARRAY [0..2] OF REAL
GET
aIMU2Acceleration := fbAccelerationSensor2.aAccelerationValues;
END_GET
END_PROPERTY

METHOD PRIVATE doSetOperationMode
VAR
END_VAR
VAR_INPUT
END_VAR
IF nGCControlOption.0 THEN
	fbGuidanceControllerXMC1.eOperationMode := GCControllerMode.CurrentControlled;
	fbGuidanceControllerXMC2.eOperationMode := GCControllerMode.CurrentControlled;
	fbGuidanceControllerXMC3.eOperationMode := GCControllerMode.CurrentControlled;
	fbGuidanceControllerXMC4.eOperationMode := GCControllerMode.CurrentControlled;
	
	bEnableIControl := TRUE;
	bEnablePControl := FALSE;
END_IF

IF nGCControlOption.1 THEN
	fbGuidanceControllerXMC1.eOperationMode := GCControllerMode.ForceControlled;
	fbGuidanceControllerXMC2.eOperationMode := GCControllerMode.ForceControlled;
	fbGuidanceControllerXMC3.eOperationMode := GCControllerMode.ForceControlled;
	fbGuidanceControllerXMC4.eOperationMode := GCControllerMode.ForceControlled;
	
	bEnableIControl := FALSE;
	bEnablePControl := TRUE;
END_IF
END_METHOD

PROPERTY eCondition : HighLevelCondition
GET
IF eActivationStatus = ActivationStatus.Disabled THEN
	eCondition := HighLevelCondition.SLEEP;
ELSE
	IF fbAccelerationSensor1.eCondition = SubLevelCondition.RUN AND fbAccelerationSensor2.eCondition = SubLevelCondition.RUN AND fbGuidanceControllerXMC1.eCondition = SubLevelCondition.RUN AND fbGuidanceControllerXMC2.eCondition = SubLevelCondition.RUN AND fbGuidanceControllerXMC3.eCondition = SubLevelCondition.RUN AND fbGuidanceControllerXMC4.eCondition = SubLevelCondition.RUN THEN
		eCondition := HighLevelCondition.RUN;
	ELSE
		eCondition := HighLevelCondition.INIT;
	END_IF
END_IF
END_GET
END_PROPERTY

PROPERTY nErrorID : UDINT
GET
VAR
	nErrorBitsIMU1 : UDINT;
	nErrorBitsIMU2 : UDINT;
	nErrorBitsGCXMC1 : UDINT;
	nErrorBitsGCXMC2 : UDINT;
	nErrorBitsGCXMC3 : UDINT;
	nErrorBitsGCXMC4 : UDINT;
END_VAR
nErrorBitsIMU1 := fbAccelerationSensor1.nErrorID;
nErrorBitsIMU2 := fbAccelerationSensor2.nErrorID;
nErrorBitsGCXMC1 := fbGuidanceControllerXMC1.nErrorID;
nErrorBitsGCXMC2 := fbGuidanceControllerXMC2.nErrorID;
nErrorBitsGCXMC3 := fbGuidanceControllerXMC3.nErrorID;
nErrorBitsGCXMC4 := fbGuidanceControllerXMC4.nErrorID;

//ErrorBits
nErrorID.0 := nErrorBitsIMU1.0;
nErrorID.1 := nErrorBitsIMU1.1;
nErrorID.2 := nErrorBitsIMU2.0;
nErrorID.3 := nErrorBitsIMU2.1;
nErrorID.4 := nErrorBitsGCXMC1.0;
nErrorID.5 := nErrorBitsGCXMC1.1;
nErrorID.6 := nErrorBitsGCXMC1.2;
nErrorID.7 := nErrorBitsGCXMC2.0;
nErrorID.8 := nErrorBitsGCXMC2.1;
nErrorID.9 := nErrorBitsGCXMC2.2;
nErrorID.10 := nErrorBitsGCXMC3.0;
nErrorID.11 := nErrorBitsGCXMC3.1;
nErrorID.12 := nErrorBitsGCXMC3.2;
nErrorID.13 := nErrorBitsGCXMC4.0;
nErrorID.14 := nErrorBitsGCXMC4.1;
nErrorID.15 := nErrorBitsGCXMC4.2;
END_GET
END_PROPERTY

END_FUNCTION_BLOCK

// ---- POUs/Guidance/FB_AccelerationSensor.TcPOU
FUNCTION_BLOCK FB_AccelerationSensor IMPLEMENTS ITF_SubSystem
VAR_OUTPUT
	aAccelerationValues : ARRAY [0..2] OF REAL;
END_VAR
VAR_IN_OUT
	stRS232Inputs : EL6inData22B;
	stRS232Outputs : EL6outData22B;
END_VAR
VAR
	//Local
	fbEL6001	: FB_SerialComRS232;
	fPacketRate : REAL := 0;
	bStartPacketCount : BOOL;
	
	fbTimer : TON;
	fbReset : TON;
	fbTrigger : R_TRIG;
	nCounter1 : UDINT;
	nCounter2 : UDINT;
	aPackets : ARRAY [0..9] OF UDINT;
	i : UDINT := 0;
	nSum : UDINT := 0;
	bTrigger : BOOL := FALSE;
	
	//ErrorBits
	bCommunicationError : BIT;
	bOutOfRange : BIT;
END_VAR
VAR CONSTANT
	fGravitationalAcceleration : REAL := 9.81;  					//in m/s^2
END_VAR

fbEL6001(stEL6001In:=stRS232Inputs, stEL6001Out:=stRS232Outputs);

aAccelerationValues := fbEL6001.aAcceleration;

doPacketCount();

METHOD PRIVATE doCheckRange : BOOL
VAR_INPUT
	aValues : ARRAY [0..2] OF REAL;
	fMax : REAL;
END_VAR
IF ABS(aValues[0]) <= fMax AND ABS(aValues[1]) <= fMax AND ABS(aValues[2]) <= fMax THEN
	doCheckRange := TRUE;
ELSE
	doCheckRange := FALSE;
END_IF
END_METHOD

METHOD PRIVATE doPacketCount
VAR_INPUT
END_VAR
fbTimer(IN := bStartPacketCount, PT := T#1S);
fbTrigger(CLK := fbTimer.IN);

IF fbTrigger.Q THEN
	nCounter1 := fbEL6001.nReceiveCounter;
END_IF

IF fbTimer.Q THEN
	nCounter2 := fbEL6001.nReceiveCounter;
	aPackets[i] := nCounter2 - nCounter1;
	nSum := nSum + aPackets[i];
	i := i + 1;
	bTrigger := TRUE;
	bStartPacketCount := FALSE;
END_IF

IF i = 10 THEN
	bTrigger := FALSE;
	fPacketRate := (UDINT_TO_REAL(nSum) / UDINT_TO_REAL(i));
	i := 0;
	nSum := 0;
	
	bStartPacketCount := TRUE;
END_IF

fbReset(IN := bTrigger, PT := T#3S);
IF fbReset.Q THEN
	bStartPacketCount := TRUE;
	bTrigger := FALSE;
END_IF
END_METHOD

PROPERTY PUBLIC eCondition : SubLevelCondition
GET
IF nErrorID <> 0 THEN
	eCondition := SubLevelCondition.ERROR;
ELSE
	eCondition := SubLevelCondition.RUN;
END_IF
END_GET
END_PROPERTY

PROPERTY PUBLIC nErrorID : UDINT
GET
IF fbEL6001.eReceiveErrorID <> COMERROR_NOERROR THEN
	bCommunicationError := TRUE;
ELSE
	bCommunicationError := FALSE;
END_IF

bOutOfRange := NOT doCheckRange(aValues:=aAccelerationValues, fMax:=2*fGravitationalAcceleration);


nErrorID.0 := bCommunicationError;
nErrorID.1 := bOutOfRange;
END_GET
END_PROPERTY

END_FUNCTION_BLOCK

// ---- POUs/Guidance/AccelerationSensor/FB_SerialComRS232.TcPOU
FUNCTION_BLOCK FB_SerialComRS232
VAR_IN_OUT
	stEL6001In : EL6inData22B;
	stEL6001Out : EL6outData22B;
END_VAR
VAR_OUTPUT
	aAcceleration : ARRAY [0..2] OF REAL;
	eReceiveErrorID	: ComError_t;
	nReceiveCounter	: UDINT;
END_VAR
VAR
	//Receive Buffer
	fbEL6001Ctrl		: SerialLineControl;
	TxBuffer	: ComBuffer;
	RxBuffer	: ComBuffer;
	//Receive Data
	fbReceive		: ReceiveData;
	nPrefix : ARRAY[0..1] OF BYTE;
	aReceiveData : ARRAY [0..15] OF BYTE;
	nPacketID : BYTE := 37;
	nPacketLength : BYTE := 12;	
	
	nCRC : WORD;
	nCheckCRC : WORD;
	nPointerCRC : POINTER TO WORD;
	aCRC : ARRAY [0..1] OF BYTE;	
	aDataArray : ARRAY[0..11] OF BYTE;
	i : USINT;
	aAccX : ARRAY [0..3] OF BYTE;
	aAccY : ARRAY [0..3] OF BYTE;
	aAccZ : ARRAY [0..3] OF BYTE;
	fPointerToX : POINTER TO REAL;
    fAccX : REAL;
	fPointerToY : POINTER TO REAL;
    fAccY : REAL;
	fPointerToZ : POINTER TO REAL;
    fAccZ : REAL;
END_VAR

fbEL6001Ctrl(
	Mode:= SERIALLINEMODE_EL6_22B, 
	pComIn:= ADR(stEL6001In), 
	pComOut:= ADR(stEL6001Out), 
	SizeComIn:= SIZEOF(stEL6001In), 
	Error=> , 
	ErrorID=> , 
	TxBuffer:= TxBuffer, 
	RxBuffer:= RxBuffer);

nPrefix[0] := nPacketID;
nPrefix[1] := nPacketLength;

fbReceive(
	RXbuffer:= RxBuffer,
	pPrefix := ADR(nPrefix),
	LenPrefix := 2,
	pReceiveData := ADR(aReceiveData),
	SizeReceiveData  := 16,								
	Error => eReceiveErrorID,
	DataReceived=>);
		
IF fbReceive.DataReceived THEN							
	nReceiveCounter := nReceiveCounter + 1;
END_IF

doCRC16Check();
doCalculateAccValues();

METHOD PRIVATE doCalculateAccValues
VAR_INPUT
END_VAR
IF nCheckCRC = nCRC THEN
	aAccX[0] := aReceiveData[4];
	aAccX[1] := aReceiveData[5];
	aAccX[2] := aReceiveData[6];
	aAccX[3] := aReceiveData[7];
	fPointerToX := ADR(aAccX);
	fAccX := fPointerToX^;
	
	aAccY[0] := aReceiveData[8];
	aAccY[1] := aReceiveData[9];
	aAccY[2] := aReceiveData[10];
	aAccY[3] := aReceiveData[11];
	fPointerToY := ADR(aAccY);
	fAccY := fPointerToY^;
	
	aAccZ[0] := aReceiveData[12];
	aAccZ[1] := aReceiveData[13];
	aAccZ[2] := aReceiveData[14];
	aAccZ[3] := aReceiveData[15];
	fPointerToZ := ADR(aAccZ);
	fAccZ := fPointerToZ^;
END_IF

aAcceleration[0] := fAccX;
aAcceleration[1] := fAccY;
aAcceleration[2] := fAccZ;
END_METHOD

METHOD PRIVATE doCRC16Check : BOOL
VAR_INPUT
END_VAR
FOR i:=0 TO 11 DO
	aDataArray[i] := aReceiveData[i+4];
END_FOR


nCRC := F_DATA_TO_CRC16_CCITT(
	pData := ADR(aDataArray),
	cbData := BYTE_TO_UDINT(nPacketLength),
	crc := 16#FFFF);

aCRC[0] := aReceiveData[2];
aCRC[1] := aReceiveData[3];
nPointerCRC := ADR(aCRC);
nCheckCRC := nPointerCRC^;
END_METHOD

END_FUNCTION_BLOCK

// ---- POUs/Guidance/FB_GuidanceController.TcPOU
FUNCTION_BLOCK FB_GuidanceController IMPLEMENTS ITF_SubSystem
VAR_INPUT
	eOperationMode : GCControllerMode;
	bActive : BOOL;
	
	fDesiredDeviationFromCenterLine : REAL;
	fActualYDistance : REAL;
	fActualYAcceleration : REAL;
	fActualCurrent	: REAL;
END_VAR
VAR_OUTPUT
	fNewReferenceValueForCurrent : REAL;
	fNewRefrenceValueForForce : REAL;
	fNewreferenceValueForVoltage : REAL;
END_VAR
VAR
	//ErrorBits
	bCurrentOutOfRange : BOOL;
	bVoltageOutOfRange : BOOL;
	bForceOutOfRange	: BOOL;
END_VAR

CASE eOperationMode OF
	GCControllerMode.CurrentControlled:
		IF bActive THEN //Implement Method with Controller Structure
			doCalculateNewReferenceValueForCurrent(fDesiredDeviationFromCenterLine := fDesiredDeviationFromCenterLine,
													fActualYDistance := fActualYDistance,
													fActualYAcceleration := fActualYAcceleration,
													fActualCurrent := fActualCurrent);
		ELSE
			fNewReferenceValueForCurrent := 0;
			fNewRefrenceValueForForce := 0;
			fNewreferenceValueForVoltage := 0;
		END_IF

	GCControllerMode.ForceControlled:
		IF bActive THEN //Implement Method with Controller Structure
			doCalculateNewReferenceValueForCurrent(fDesiredDeviationFromCenterLine := fDesiredDeviationFromCenterLine,
													fActualYDistance := fActualYDistance,
													fActualYAcceleration := fActualYAcceleration,
													fActualCurrent := fActualCurrent);
		ELSE
			fNewReferenceValueForCurrent := 0;
			fNewRefrenceValueForForce := 0;	
			fNewreferenceValueForVoltage := 0;														
		END_IF
END_CASE

METHOD PRIVATE doCalculateNewReferenceValueForCurrent
VAR_INPUT
	fDesiredDeviationFromCenterLine : REAL;
	fActualYDistance : REAL;
	fActualYAcceleration : REAL;
	fActualCurrent	: REAL;
END_VAR
fNewReferenceValueForCurrent := 0;
fNewRefrenceValueForForce := 0;
fNewreferenceValueForVoltage := 0;
END_METHOD

METHOD PRIVATE doCalculateNewReferenceValueForCurrentandForce
VAR_INPUT
	fDesiredDeviationFromCenterLine : REAL;
	fActualYDistance : REAL;
	fActualYAcceleration : REAL;
	fActualCurrent	: REAL;
END_VAR
fNewReferenceValueForCurrent := 0;
fNewRefrenceValueForForce := 0;
fNewreferenceValueForVoltage := 0;
END_METHOD

PROPERTY PUBLIC eCondition : SubLevelCondition
GET
IF nErrorID <> 0 THEN
	eCondition := SubLevelCondition.ERROR;
ELSE
	eCondition := SubLevelCondition.RUN;
END_IF
END_GET
END_PROPERTY

PROPERTY PUBLIC nErrorID : UDINT
GET
//RangeAbfrage to be implemented
bCurrentOutOfRange := FALSE;
bVoltageOutOfRange := FALSE;
bForceOutOfRange := FALSE;

nErrorID.0 := bCurrentOutOfRange;
nErrorID.1 := bVoltageOutOfRange;
nErrorID.2 := bForceOutOfRange;
END_GET
END_PROPERTY

END_FUNCTION_BLOCK

// ---- POUs/ErrorHandling/FB_SafetyCounter.TcPOU
FUNCTION_BLOCK FB_SafetyCounter
VAR_INPUT
	bReset : BOOL;
END_VAR
VAR_OUTPUT
	nSafetyCounter : UDINT;
END_VAR
VAR
	nSafetyCounterOC 	: UDINT;
	nSafetyCounterXMC1 	: UDINT;
	nSafetyCounterXMC2 	: UDINT;
	nSafetyCounterXMC3 	: UDINT;
	nSafetyCounterXMC4 	: UDINT;
	

	fbTimeoutOC : TON := (PT := PRG_ErrorHandling.tSafetyCounterTimeout);
	fbTimeoutXMC1 : TON := (PT := PRG_ErrorHandling.tSafetyCounterTimeout);
	fbTimeoutXMC2 : TON := (PT := PRG_ErrorHandling.tSafetyCounterTimeout);
	fbTimeoutXMC3 : TON := (PT := PRG_ErrorHandling.tSafetyCounterTimeout);
	fbTimeoutXMC4 : TON := (PT := PRG_ErrorHandling.tSafetyCounterTimeout);
	fbTimeoutEtherCAT : TON := (PT := PRG_ErrorHandling.tSafetyCounterTimeout);
	
	fbFrameCounter : FB_EcMasterFrameStatistic;
	bCount : BOOL;
	fFramesPerSecond : LREAL;
	
	//ErrorBits
	bNoConnectionToOC : BOOL;
	bNoConnectionToXMC1 : BOOL;
	bNoConnectionToXMC2 : BOOL;
	bNoConnectionToXMC3 : BOOL;
	bNoConnectionToXMC4 : BOOL;
	bNoEtherCATConnection : BOOL;
END_VAR
VAR CONSTANT
	nCounterMax : UDINT := 4294967295;
END_VAR

IF NOT PRG_ErrorHandling.nTestMode.1 THEN
	doEtherCATFrameCount();
END_IF

nSafetyCounter := nSafetyCounter + 1;
IF nSafetyCounter = nCounterMax THEN
	nSafetyCounter := 0;
END_IF

//OC
IF NOT PRG_ErrorHandling.nTestMode.0 THEN
	IF PRG_MainController.stOperationControlCommands.nSafetyCounterOC <> nSafetyCounterOC THEN
		nSafetyCounterOC := PRG_MainController.stOperationControlCommands.nSafetyCounterOC;
		fbTimeoutOC(IN := FALSE);
		bNoConnectionToOC := FALSE;
	ELSE
		fbTimeoutOC(IN := NOT bReset);
		bNoConnectionToOC := FALSE;
		IF fbTimeoutOC.Q THEN
			bNoConnectionToOC := TRUE;
		END_IF
	END_IF
END_IF

//XMC1
IF NOT PRG_ErrorHandling.nTestMode.2 THEN
	IF PRG_MainController.stXMCCommands.nSafetyCounterXMC1 <> nSafetyCounterXMC1 THEN
		nSafetyCounterXMC1 := PRG_MainController.stXMCCommands.nSafetyCounterXMC1;
		fbTimeoutXMC1(IN := FALSE);
		bNoConnectionToXMC1 := FALSE;
	ELSE
		fbTimeoutXMC1(IN:= NOT bReset);
		bNoConnectionToXMC1 := FALSE;
		IF fbTimeoutXMC1.Q THEN
			bNoConnectionToXMC1 := TRUE;
		END_IF
	END_IF
END_IF

//XMC2
IF NOT PRG_ErrorHandling.nTestMode.3 THEN
	IF PRG_MainController.stXMCCommands.nSafetyCounterXMC2 <> nSafetyCounterXMC2 THEN
		nSafetyCounterXMC2 := PRG_MainController.stXMCCommands.nSafetyCounterXMC2;
		fbTimeoutXMC2(IN := FALSE);
		bNoConnectionToXMC2 := FALSE;
	ELSE
		fbTimeoutXMC2(IN:= NOT bReset);
		bNoConnectionToXMC2 := FALSE;
		IF fbTimeoutXMC2.Q THEN
			bNoConnectionToXMC2 := TRUE;
		END_IF
	END_IF
END_IF

//XMC3
IF NOT PRG_ErrorHandling.nTestMode.4 THEN
	IF PRG_MainController.stXMCCommands.nSafetyCounterXMC3 <> nSafetyCounterXMC3 THEN
		nSafetyCounterXMC3 := PRG_MainController.stXMCCommands.nSafetyCounterXMC3;
		fbTimeoutXMC3(IN := FALSE);
		bNoConnectionToXMC3 := FALSE;
	ELSE
		fbTimeoutXMC3(IN:= NOT bReset);
		bNoConnectionToXMC3 := FALSE;
		IF fbTimeoutXMC3.Q THEN
			bNoConnectionToXMC3 := TRUE;
		END_IF
	END_IF
END_IF

//XMC4
IF NOT PRG_ErrorHandling.nTestMode.5 THEN
	IF PRG_MainController.stXMCCommands.nSafetyCounterXMC4 <> nSafetyCounterXMC4 THEN
		nSafetyCounterXMC4 := PRG_MainController.stXMCCommands.nSafetyCounterXMC4;
		fbTimeoutXMC4(IN := FALSE);
		bNoConnectionToXMC4 := FALSE;
		fbTimeoutXMC1(IN := FALSE);
	ELSE
		fbTimeoutXMC4(IN:= NOT bReset);
		bNoConnectionToXMC4 := FALSE;
		IF fbTimeoutXMC4.Q THEN
			bNoConnectionToXMC4 := TRUE;
		END_IF
	END_IF
END_IF

METHOD PRIVATE doEtherCATFrameCount
VAR_INPUT
END_VAR
IF NOT bCount THEN
	bCount := TRUE;
	fbFrameCounter(sNetId := '5.93.125.76.4.1', bExecute := bCount, fFramesPerSecond => fFramesPerSecond);
END_IF

IF bCount THEN
	bCount := FALSE;
	fbFrameCounter(sNetId := '5.93.125.76.4.1', bExecute := bCount, fFramesPerSecond => fFramesPerSecond);
END_IF

IF fFramesPerSecond <> 0 THEN
	bNoEtherCATConnection := FALSE;
	fbTimeoutEtherCAT(IN := FALSE);
ELSE
	fbTimeoutEtherCAT(IN := NOT bReset);
	bNoEtherCATConnection := FALSE;
	IF fbTimeoutEtherCAT.Q THEN
		bNoEtherCATConnection := TRUE;
	END_IF
END_IF
END_METHOD

PROPERTY PUBLIC nErrorID : UDINT
GET
nErrorID.0 := 	bNoConnectionToOC;
nErrorID.1 :=	bNoConnectionToXMC1;
nErrorID.2 :=	bNoConnectionToXMC2;
nErrorID.3 :=	bNoConnectionToXMC3;
nErrorID.4 := 	bNoConnectionToXMC4;
nErrorID.5 :=	bNoEtherCATConnection;
END_GET
END_PROPERTY

END_FUNCTION_BLOCK
